(* PLC project Unnamed, Unknown Unnamed 1 *)
(* stored: creationDateTime 2023-03-10T10:37:17, modificationDateTime 2023-03-15T15:56:42 *)

(* ISBN: 978-3-8085-3450-2, Klimaanlage *)
FUNCTION_BLOCK Air_Condition_Control
  VAR_INPUT
    IN1 : BOOL;
    IN2 : BOOL;
    IN3 : BOOL;
    IN4 : BOOL;
    IN5 : BOOL;
    IN6 : BOOL;
    IN7 : BOOL;
    IN8 : BOOL;
    IN9 : BOOL;
  END_VAR
  VAR_OUTPUT
    OUT1 : BOOL;
    OUT2 : BOOL;
  END_VAR
  VAR
    RS0 : RS;
  END_VAR

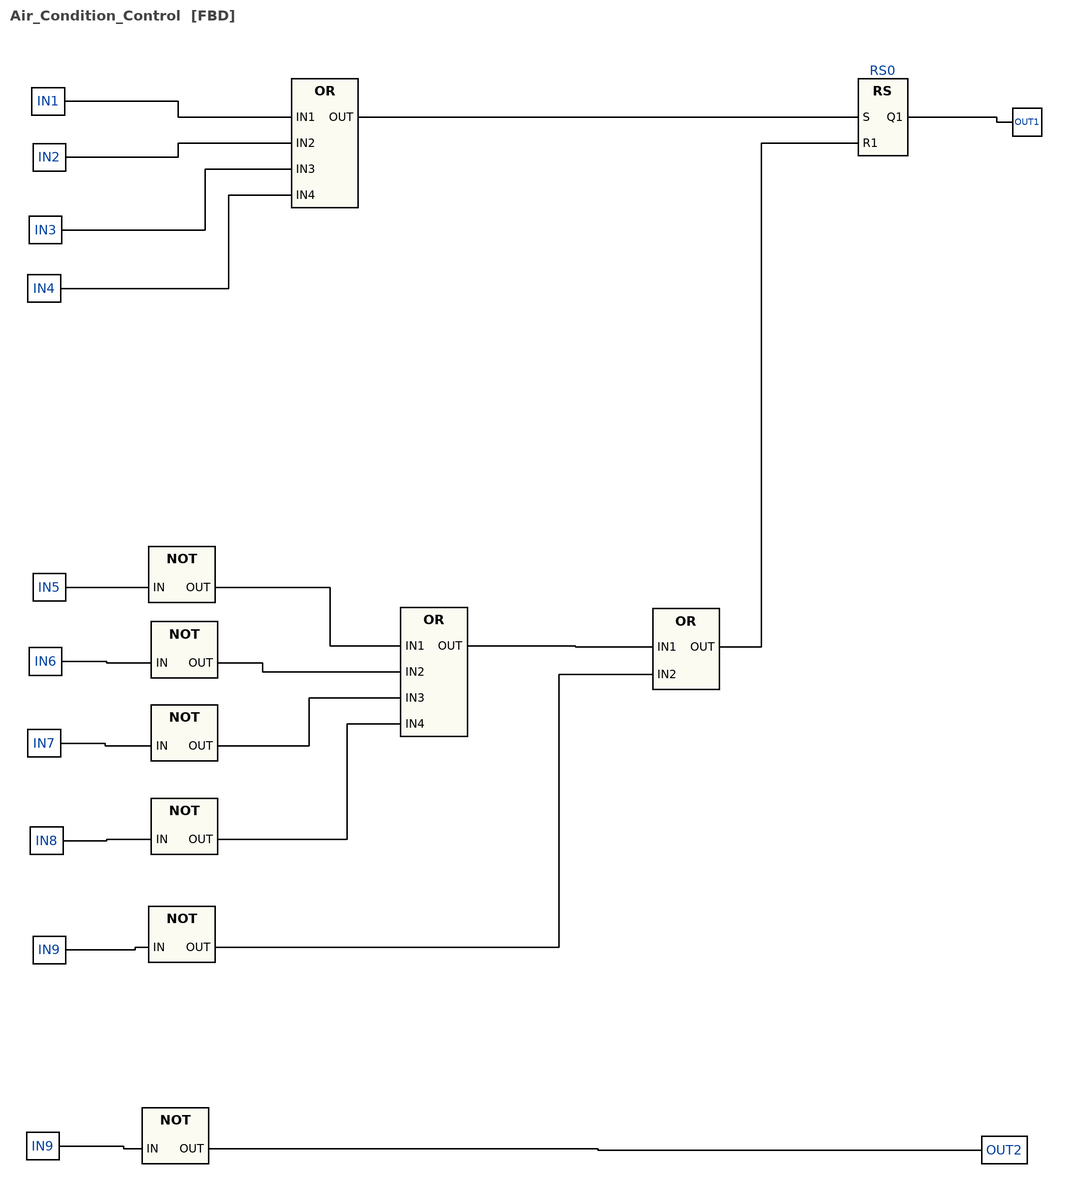
(* FBD diagram, written out as Structured Text *)
RS0(S := IN1 OR IN2 OR IN3 OR IN4, R1 := NOT IN5 OR NOT IN6 OR NOT IN7 OR NOT IN8 OR NOT IN9);
OUT1 := RS0.Q1;
OUT2 := NOT IN9;
END_FUNCTION_BLOCK

CONFIGURATION config
  RESOURCE resource1 ON PLC
  END_RESOURCE
END_CONFIGURATION
